INTERFACE I_Door

METHOD PUBLIC m_Close : BOOL
END_METHOD

METHOD PUBLIC m_Open : BOOL
END_METHOD

METHOD PUBLIC m_Reset : BOOL
END_METHOD

METHOD PUBLIC m_Stop : BOOL
END_METHOD

{attribute 'monitoring':='call'}
PROPERTY PUBLIC p_bStaIsClosed : BOOL
GET
END_GET
END_PROPERTY

{attribute 'monitoring':='call'}
PROPERTY PUBLIC p_bStaIsClosing : BOOL
GET
END_GET
END_PROPERTY

{attribute 'monitoring':='call'}
PROPERTY PUBLIC p_bStaIsOpened : BOOL
GET
END_GET
END_PROPERTY

{attribute 'monitoring':='call'}
PROPERTY PUBLIC p_bStaIsOpening : BOOL
GET
END_GET
END_PROPERTY

END_INTERFACE

(* stored: Version 1.1.0.1, ProductVersion 3.1.4024.12
   Itf I_Door: Id {7f72806e-1a4d-4a0f-936c-bcb2882fc369}
   Folder Methods: Id {8f726fdf-c22c-4ce9-9c80-969f6e8d7f6d}
   Folder Properties: Id {7896c925-8494-43ef-976f-5dcd6349882e}
   Method m_Close: Id {7d25f223-1aed-4fba-93f7-afa16a294a93}
   Method m_Open: Id {41dc07a6-74ce-485b-b57c-2bc432648dfa}
   Method m_Reset: Id {10b9821f-e854-465e-b13d-3b3987fe37c1}
   Method m_Stop: Id {93faa1ac-c7dc-4632-9d6b-ba891a448322}
   Property p_bStaIsClosed: Id {0e698f60-99c2-43ca-9697-801888d79762}
   Get Get: Id {0720a712-6396-48c3-af32-35cfaed3e694}
   Property p_bStaIsClosing: Id {da905841-3391-4d5d-a9a8-39af8abf8d8c}
   Get Get: Id {9a7c56bb-9e7e-4cd7-aa78-1f44f5d8efea}
   Property p_bStaIsOpened: Id {467b5270-27bc-48f7-996b-3a5e03afe752}
   Get Get: Id {a6276f68-23b4-4548-b5dc-07546461302e}
   Property p_bStaIsOpening: Id {2a8e4a6a-d82e-438c-8ddb-eb3cef242c14}
   Get Get: Id {811a8b45-4f74-4593-99a5-10997a3017ab} *)
